(* IEC 61131-3 sources: test/Class/Sfc_Transition_Base, 1 file *)

(* ---- Sfc_Transition_Base.st ---- *)
(*!
<Class
	Name               = "Sfc_Transition_Base"
	Revision           = "1.2"
	RealtimeTask       = "false"
	CyclicTask         = "false"
	BackgroundTask     = "false"
	Sigmatek           = "true"
	OSInterface        = "false"
	HighPriority       = "false"
	Automatic          = "false"
	UpdateMode         = "Prescan"
	SharedCommandTable = "true"
	Objectsize         = "(284,120)"
	Comment            = "Base class for transitions.">
	<Channels>
		<Server Name="TransitionItf" Visualized="false" Initialize="false" WriteProtected="false" Retentive="false" Comment="Interface to the transition class.&#13;&#10;&#13;&#10;Preceeding steps use this server to evaluate the transition."/>
		<Client Name="GetParentPtr" Required="true" Internal="false" Comment="Helper client for optaining a&#13;&#10;pointer to the parent SFC class."/>
		<Client Name="NextStep" Required="false" Internal="false" Comment="Client for activating following steps."/>
		<Client Name="PrevStep" Required="false" Internal="false" Comment="Client for disabling preceeding steps."/>
	</Channels>
	<RevDoku>
		<Owner Company="Sigmatek GmbH &amp; KG" Author="LesMax"/>
		<Dokumentation Revision="1.2" Date="2013-10-17" Author="LesMax" Company="Sigmatek GmbH &amp; KG" Description="Transitions now obtain a pointer to the&#13;&#10;parent Sfc class at initialisation."/>
		<Dokumentation Revision="1.1" Date="2013-10-14" Author="LesMax" Company="Sigmatek GmbH &amp; KG" Description="IOs of transitions can now be automatically&#13;&#10;written by setting the AutoWrite Property"/>
	</RevDoku>
</Class>
*)
Sfc_Transition_Base : CLASS
  //Servers:
	TransitionItf 	: SvrChCmd_DINT;
  //Clients:
	PrevStep 	: CltCh_DINT;
	NextStep 	: CltCh_DINT;
	GetParentPtr 	: CltCh_UDINT;
  //Variables:
  //Functions:

	FUNCTION VIRTUAL GLOBAL Init;

	FUNCTION VIRTUAL Condition
		VAR_OUTPUT
			Result 	: DINT;
		END_VAR;

	FUNCTION CheckTransition
		VAR_OUTPUT
			Result 	: DINT;
		END_VAR;

	FUNCTION VIRTUAL OnReadInternalVariables;

	FUNCTION VIRTUAL OnWriteInternalVariables;

	FUNCTION VIRTUAL GLOBAL TransitionItf::Read
		VAR_OUTPUT
			output (EAX) 	: DINT;
		END_VAR;
  //Tables:
	FUNCTION @STD
		VAR_OUTPUT
			ret_code	: CONFSTATES;
		END_VAR;
	FUNCTION GLOBAL TAB @CT_;
END_CLASS;

FUNCTION VIRTUAL GLOBAL Sfc_Transition_Base::TransitionItf::Read
	VAR_OUTPUT
		output (EAX) 	: DINT;
	END_VAR

	output := CheckTransition();

END_FUNCTION

FUNCTION Sfc_Transition_Base::CheckTransition
	VAR_OUTPUT
		Result 	: DINT;
	END_VAR

  // Read all connected internal variable servers
  OnReadInternalVariables();

  // Check if the condition is met.
  if Condition() = true then

    // Transition condition is met.
    Result := 1;

    // Deactivate the previous step.
    PrevStep.Write(input:=0);

    // Activate the next step.
    NextStep.Write(input:=1);

  else

    // Transition condition is not met
    Result := 0;

  end_if;

  // Write all connected internal variable servers
  OnWriteInternalVariables();

END_FUNCTION

// Overridable for User Conditions
FUNCTION VIRTUAL Sfc_Transition_Base::Condition
	VAR_OUTPUT
		Result 	: DINT;
	END_VAR

  // Default condition is never met.
  Result := false;

END_FUNCTION

// Overrideable for reading connected internal variable servers
FUNCTION VIRTUAL Sfc_Transition_Base::OnReadInternalVariables

END_FUNCTION

// Overrideable for writing connected internal variable servers
FUNCTION VIRTUAL Sfc_Transition_Base::OnWriteInternalVariables

END_FUNCTION

FUNCTION VIRTUAL GLOBAL Sfc_Transition_Base::Init

  if _FirstScan then

    GetParentPtr := GetParentPtr.Read();

  end_if;

END_FUNCTION
